Yaskawa INFORM job: neg_x_0.JBI

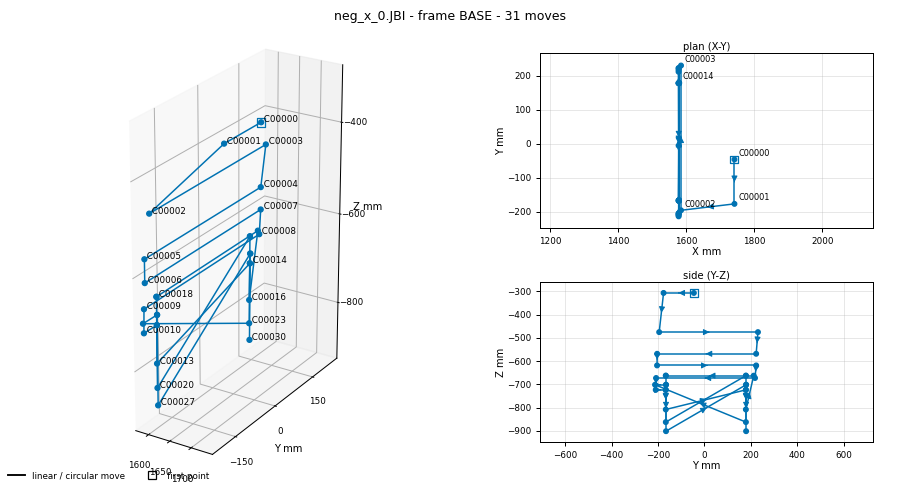
[picture p0: tool path of neg_x_0.JBI in frame BASE, 31 of 33 moves have a stored position in this frame; points joined in program order, loops and branches not executed]
/JOB
//NAME neg_x_0
//POS
///NPOS 31,0,31,0,0,0
///TOOL 0
///POSTYPE BASE
///RECTAN
///RCONF 0,0,0,0,0,0,0,0,0,0,0,0,0,0,0,0,0,0,0,0,0,0,0,0
C00000=1741.381590,-45.669052,-306.303009,180.000000,-89.999999,0.000000
C00001=1741.381590,-176.207052,-306.303009,180.000000,-89.999999,0.000000
C00002=1584.353544,-195.083398,-475.055618,180.000000,-89.999999,0.000000
C00003=1584.353544,230.369602,-475.055618,180.000000,-89.999999,0.000000
C00004=1577.352926,222.596301,-568.404381,180.000000,-89.999999,0.000000
C00005=1577.352926,-203.885699,-568.404381,180.000000,-89.999999,0.000000
C00006=1577.342619,-204.154645,-618.577970,180.000000,-89.999999,0.000000
C00007=1577.342619,222.705355,-618.577970,180.000000,-89.999999,0.000000
C00008=1577.184028,217.687895,-672.678435,180.000000,-89.999999,0.000000
C00009=1577.184028,-208.285505,-672.678435,180.000000,-89.999999,0.000000
C00010=1577.159099,-210.002270,-723.795090,180.000000,-89.999999,0.000000
C00011=1578.247563,-166.683270,-723.795090,180.000000,-89.999999,0.000000
C00012=1578.247563,-166.683270,-723.795090,180.000000,-89.999999,0.000000
C00013=1577.159099,-166.683378,-808.325036,180.000000,-60.000000,0.000000
C00014=1578.647563,178.328730,-723.795090,180.000000,-89.999999,0.000000
C00015=1578.647563,178.328730,-723.795090,180.000000,-89.999999,0.000000
C00016=1577.159099,178.328629,-808.325036,180.000000,-60.000000,0.000000
C00017=1577.106028,212.089598,-662.606578,180.000000,-60.000000,0.000000
C00018=1578.194492,-166.547702,-662.606578,180.000000,-60.000000,0.000000
C00019=1578.194492,-166.547702,-662.606578,180.000000,-60.000000,0.000000
C00020=1577.106028,-166.547810,-862.606578,180.000000,-60.000000,0.000000
C00021=1578.594492,178.464298,-662.606578,180.000000,-60.000000,0.000000
C00022=1578.594492,178.464298,-662.606578,180.000000,-60.000000,0.000000
C00023=1577.106028,178.464197,-862.606578,180.000000,-60.000000,0.000000
C00024=1577.407452,-212.883838,-701.853352,180.000000,-60.000000,0.000000
C00025=1578.495916,-165.712838,-701.853352,180.000000,-60.000000,0.000000
C00026=1578.495916,-165.712838,-701.853352,180.000000,-60.000000,0.000000
C00027=1577.407452,-165.712946,-901.853352,180.000000,-60.000000,0.000000
C00028=1578.895916,179.299162,-701.853352,180.000000,-60.000000,0.000000
C00029=1578.895916,179.299162,-701.853352,180.000000,-60.000000,0.000000
C00030=1577.407452,179.299061,-901.853352,180.000000,-60.000000,0.000000
///POSTYPE PULSE
///PULSE
EX000=92160
///POSTYPE PULSE
///PULSE
EC00000=92160
EC00001=92160
EC00002=92160
EC00003=92160
EC00004=92160
EC00005=92160
EC00006=92160
EC00007=92160
EC00008=92160
EC00009=92160
EC00010=92160
EC00011=92160
EC00012=92160
EC00013=92160
EC00014=92160
EC00015=92160
EC00016=92160
EC00017=92160
EC00018=92160
EC00019=92160
EC00020=92160
EC00021=92160
EC00022=92160
EC00023=92160
EC00024=92160
EC00025=92160
EC00026=92160
EC00027=92160
EC00028=92160
EC00029=92160
EC00030=92160
//INST
///DATE 2023/06/26 11:09
///ATTR SC,RW,RJ
////FRAME BASE
///GROUP1 RB1,ST1
NOP
MOVJ P009 EX000 VJ=15.00
MOVJ C00000 EC00000 VJ=15.0
CALL JOB:SPYON
MOVL C00001 EC00001 V=150.0
MOVL C00002 EC00002 V=150.0
MOVL C00003 EC00003 V=150.0
MOVL C00004 EC00004 V=150.0
MOVL C00005 EC00005 V=150.0
MOVL C00006 EC00006 V=150.0
MOVL C00007 EC00007 V=150.0
MOVL C00008 EC00008 V=150.0
MOVL C00009 EC00009 V=150.0
MOVL C00010 EC00010 V=150.0
CALL JOB:SPYOF
MOVL C00011 EC00011 V=150.0
CALL JOB:SPYON
MOVL C00012 EC00012 V=150.0
CALL JOB:SPYOF
MOVL C00013 EC00013 V=150.0
MOVL C00014 EC00014 V=150.0
CALL JOB:SPYON
MOVL C00015 EC00015 V=150.0
CALL JOB:SPYOF
MOVL C00016 EC00016 V=150.0
CALL JOB:SPYON
MOVL C00017 EC00017 V=150.0
CALL JOB:SPYOF
MOVL C00018 EC00018 V=150.0
CALL JOB:SPYON
MOVL C00019 EC00019 V=150.0
CALL JOB:SPYOF
MOVL C00020 EC00020 V=150.0
MOVL C00021 EC00021 V=150.0
CALL JOB:SPYON
MOVL C00022 EC00022 V=150.0
CALL JOB:SPYOF
MOVL C00023 EC00023 V=150.0
CALL JOB:SPYON
MOVL C00024 EC00024 V=150.0
CALL JOB:SPYOF
MOVL C00025 EC00025 V=150.0
CALL JOB:SPYON
MOVL C00026 EC00026 V=150.0
CALL JOB:SPYOF
MOVL C00027 EC00027 V=150.0
MOVL C00028 EC00028 V=150.0
CALL JOB:SPYON
MOVL C00029 EC00029 V=150.0
CALL JOB:SPYOF
MOVL C00030 EC00030 V=150.0
CALL JOB:SPYOF
MOVJ P009 VJ=15.00
END
